{attribute 'GeneratedUsingTerminal: AT2050-0500-0019'}
{attribute addProperty BoxType "AT2050-0500-0019"}
{attribute addProperty Id "A_0094_AT2021_5250_0018_AT2021_5250AT2021_33A3DF1B80"}
{attribute addProperty CRC "363048559"}
{attribute addProperty Size "80"}
TYPE A_0050_AT2050_0500_0019_15A3AE6F EXTENDS AT2050_2EA6C9BF :
STRUCT
	{attribute addProperty Name "A_0094_AT2021_5250_0018_AT2021_5250"}
	{attribute addProperty PreviousPort "A_0050(AT2050-0500-0019) : B"}
	A_0094_AT2021_5250_0018_AT2021_5250 : AT2021_33A3DF1B;
END_STRUCT
END_TYPE

(* stored: Version 1.2.0.0, ProductVersion 3.1.4024.9
   DUT A_0050_AT2050_0500_0019_15A3AE6F: Id {4d195701-da41-4185-a074-5130a42c1a16} *)
